FUNCTION F_HE_SATT_MaterialToMaterialFormula : T_MaxString
VAR_INPUT
    eMaterial : E_HE_SATT_FilterMaterial;
END_VAR


CASE eMaterial OF
    E_HE_SATT_FilterMaterial.Diamond:
        F_HE_SATT_MaterialToMaterialFormula := 'C';
        
    E_HE_SATT_FilterMaterial.Germanium:
        F_HE_SATT_MaterialToMaterialFormula := 'Ge';
        
    E_HE_SATT_FilterMaterial.Silicon:
        F_HE_SATT_MaterialToMaterialFormula := 'Si';
        
    ELSE
        F_HE_SATT_MaterialToMaterialFormula := TO_STRING(eMaterial);
END_CASE

END_FUNCTION

(* stored: Version 1.1.0.1
   POU F_HE_SATT_MaterialToMaterialFormula: Id {351079bf-21c6-4c05-8134-9faa64daf259}, SpecialFunc None *)
